(* CODESYS project PI.project

Project tree, tasks and I/O mapping:
  Device : CODESYS Control for Raspberry Pi, 3S - Smart Software Solutions GmbH, version 3.5.6.0
    application Application
      libraries: Standard, * (System)
      task MainTask (cyclic, interval t#20ms, priority 1) calls PLC_PRG
      task EtherCAT_Master (cyclic, interval 4000 µs, priority 0) calls EtherCAT_Master.EtherCAT_Task [EtherCAT_Master.EtherCAT_Task]
      program PLC_PRG [ST]
      Symbols
    SoftMotion General Axis Pool
    GPIOs_A_B : GPIOs A/B, 3S - Smart Software Solutions GmbH, version 1.1.1.0
        unmapped channels: digital inputs (GPIO0..GPIO31), digital outputs (GPIO0..GPIO31)
    I²C
    SPI
    Onewire
    Camera device
      <Empty>
    EtherCAT_Master : EtherCAT Master, 3S - Smart Software Solutions GmbH, version 3.5.5.0
        settings: NetworkName = 'eth1'; SrcAddress1 = 60450; SrcAddress2 = 2158188356
      EK1100 : EK1100 EtherCAT Coupler (2A E-Bus), Beckhoff Automation GmbH, version Revision=16#00110000
          settings: StationAlias = 0; DC sync0 cycletime = 4000; DC sync1 cycletime = 4000
        EL1008 : EL1008 8Ch. Dig. Input 24V, 3ms, Beckhoff Automation GmbH, version Revision=16#00100000
            settings: StationAlias = 0; DC sync0 cycletime = 4000; DC sync1 cycletime = 4000
            input  I0 : BIT  // Input
            input  I1 : BIT  // Input
            input  I2 : BIT  // Input
            input  I3 : BIT  // Input
            unmapped channels: Input, Input, Input, Input
        EL2008 : EL2008 8Ch. Dig. Output 24V, 0.5A, Beckhoff Automation GmbH, version Revision=16#00100000
            settings: StationAlias = 0; DC sync0 cycletime = 4000; DC sync1 cycletime = 4000
            output Q0 : BIT  // Output
            output Q1 : BIT  // Output
            output Q2 : BIT  // Output
            output Q3 : BIT  // Output
            unmapped channels: Output, Output, Output, Output
        EL3062 : EL3062 2Ch. Ana. Input 0-10V, Beckhoff Automation GmbH, version Revision=16#00110000
            settings: StationAlias = 0; DC sync0 cycletime = 4000; DC sync1 cycletime = 4000
            input  AI0 : INT  // Value
            input  AI1 : INT  // Value
            unmapped channels: Status__Underrange, Status__Overrange, Status__Limit 1, Status__Limit 1, Status__Limit 2, Status__Limit 2, Status__Error, ---, ---, ---, ---, ---, ---, ---, Status__TxPDO State, Status__TxPDO Toggle, Status__Underrange, Status__Overrange, Status__Limit 1, Status__Limit 1, Status__Limit 2, Status__Limit 2, Status__Error, ---, ---, ---, ---, ---, ---, ---, Status__TxPDO State, Status__TxPDO Toggle
        EL4002 : EL4002 2Ch. Ana. Output 0-10V, 12bit, Beckhoff Automation GmbH, version Revision=16#00130000
            settings: StationAlias = 0
            output AO0 : INT  // Analog output
            unmapped channels: Analog output
        EK1110 : EK1110 EtherCAT extension, Beckhoff Automation GmbH, version Revision=16#00100000
            settings: StationAlias = 0; DC sync0 cycletime = 4000; DC sync1 cycletime = 4000
*)

// Device/Application/PLC_PRG
PROGRAM PLC_PRG
VAR
	OPC_VAL: INT;
END_VAR

Q0 := I0;
Q1 := I1;
Q2 := I2;
Q3 := I3;
AO0 := OPC_VAL;

END_PROGRAM
